PROGRAM MAIN
VAR
END_VAR

END_PROGRAM

(* stored: Version 1.1.0.1
   POU MAIN: Id {32465e2d-2260-45f4-9991-7811890b787f} *)
